INTERFACE I_MotionAxisDS402 EXTENDS I_MotionAxis

METHOD ModeOfOperation : BOOL;
VAR_INPUT
    RecentModeOfOperation : E_DS402OpMode;
END_VAR
END_METHOD

END_INTERFACE

(* stored: Version 1.1.0.1
   Itf I_MotionAxisDS402: Id {3455f02d-95d0-4a12-be21-347f31df3d3f}
   Method ModeOfOperation: Id {95fb2066-e6f8-4b6a-88d0-1139481adf13} *)
